(* Schneider Machine Expert - Basic project 09_symbols, file version 3.0.0.0 *)
(* ProjectInformations: Name=New project *)

HARDWARE
  Cpu 0: TM221CE16R
  EthernetConfiguration: NetworkName=M221, IpAllocationMode=FixedAddress, IpAddress=0.0.0.0, SubnetMask=0.0.0.0
  SerialLineConfiguration: Baud=Baud19200, Parity=ParityEven, DataBits=DataBits8, StopBits=StopBits1, PhysicalMedium=PhysicalMediumRs485, TransmissionMode=TransmissionModeModbusRtu, SlaveId=1, Addressing=SlaveAddressing
  MastTask: UsePeriodScanMode=false, PeriodScan=100
  FastTask: Period=255
  CpuBehavior: StartingMode=StartAsPreviousState, AutoSaveRamOnEeprom=true, WatchdogPeriod=250

SYMBOLS  (address, symbol, comment, settings)
  %M0       RUN_LATCH
  %C0       PART_COUNT
  %I0.0     START_PB  "Start push button"
  %Q0.0     MOTOR_RUN  "Motor contactor"

POU New POU
  (* SectionNumber=0 *)

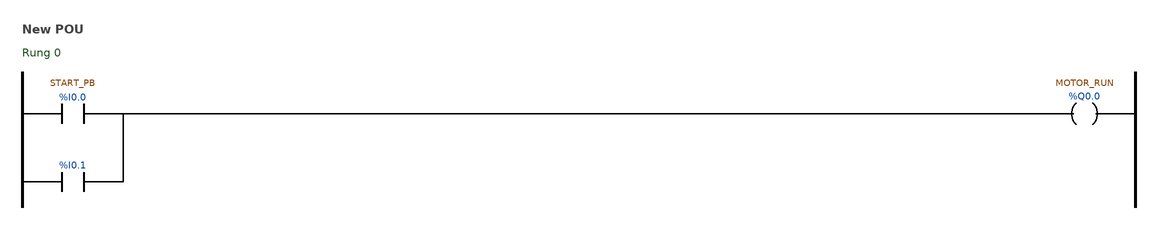

// Rung 0
  LD %I0.0                (* START_PB *)
  OR %I0.1
  ST %Q0.0                (* MOTOR_RUN *)
  // as ST:
  //   MOTOR_RUN := START_PB OR %I0.1;
